PROGRAM prgModbus
// 06.10.25 Ladestationen
VAR
	FB_LS_125 :FB_ECS_KEBA_P30:= (bEnable:= TRUE, sIPAdress:= '192.168.1.125');
	FB_LS_212 :FB_ECS_KEBA_P30:= (bEnable:= TRUE, sIPAdress:= '192.168.1.212');
	FB_LS_120 :FB_ECS_KEBA_P30:= (bEnable:= TRUE, sIPAdress:= '192.168.1.120');
END_VAR


FB_LS_125();
//FB_LS_212();
//FB_LS_120();

END_PROGRAM

(* stored: Version 1.1.0.1, ProductVersion 3.1.4024.15
   POU prgModbus: Id {c5effa87-a89a-49c4-8da2-f92b21cd7ae1}, SpecialFunc None *)
